(* IEC 61131-3 sources: eCockpitGit/test_project/src/%F%00 Library/%F%Common Functions/%F%Networking/%POU%FB_TCPMultiPlexer, 7 files *)

(* ---- %METH%acceptCycle.st ---- *)
//Called cyclicly to handle incoming connections
// |**Version**|**Author**| **Date** |**Changes**
// | 1         | NSN      | 20-05-22 | Creation
METHOD acceptCycle
VAR
	i			:WORD;
END_VAR
(*%!%__DELIMITER__%!%*)
IF S_nextClosed < S_controllersSize THEN
	//Incoming connection is accepted
	IF S_listenersSize > 0 THEN
		FOR i := 0 TO S_listenersSize - 1 DO
			S_controllers^[S_nextClosed].acceptConnection(listener:=S_listeners^[i]);
		END_FOR
	END_IF
END_IF

(* ---- %METH%closeConnection.st ---- *)
//Called to close and clean up all connections in the multiplexer
// |**Version**|**Author**| **Date** |**Changes**
// | 1         | NSN      | 20-05-22 | Creation
METHOD closeConnection
VAR
	i			:WORD;
END_VAR
(*%!%__DELIMITER__%!%*)
IF S_controllersSize > 0 THEN
	FOR i := 0 TO S_controllersSize - 1 DO
		S_controllers^[i].closeConnection();
	END_FOR
END_IF

(* ---- %METH%initialize.st ---- *)
//Initializes the tcp controller with needed values
// |**Version**|**Author**| **Date** |**Changes**
// | 1         | NSN      | 20-05-22 | Creation
METHOD initialize : SLMResult
VAR_INPUT
	controllers			:POINTER TO ARRAY[0..19] OF FB_TCPController;	//List of controllers to handle connections
	controllersSize		:WORD;											//Size of controller list
	listeners			:POINTER TO ARRAY[0..19] OF TCP.Listener;		//List of listeners to check for incoming connections
	listenersSize		:WORD;											//Size of listener list
END_VAR
VAR
	i					:WORD;
END_VAR
(*%!%__DELIMITER__%!%*)
IF controllers = 0 OR controllersSize = 0 OR listeners = 0 OR listenersSize = 0 THEN
	initialize.success					:=		FALSE;
	initialize.code						:=		ERCodes.FB_TCPMultiPlexer_initialize;
	RETURN;
END_IF
S_controllers							:=		controllers;
S_controllersSize						:=		controllersSize;
FOR i := 0 TO controllersSize - 1 DO
	S_controllers^[i].S_management		:=		THIS^;
	S_controllers^[i].S_index			:=		i;
	IF S_messageEvent <> 0 THEN
		S_controllers^[i].S_message		:=		S_messageEvent;
	END_IF
END_FOR

S_listeners								:=		listeners;
S_listenersSize							:=		listenersSize;

(* ---- %METH%messageCycle.st ---- *)
//Called cyclicly to cause messages to be processed via event system
// |**Version**|**Author**| **Date** |**Changes**
// | 1         | NSN      | 20-05-22 | Creation
METHOD messageCycle
VAR
	i			:WORD;
END_VAR
(*%!%__DELIMITER__%!%*)
IF S_controllersSize > 0 THEN
	FOR i := 0 TO S_controllersSize - 1 DO
		WHILE S_controllers^[i].readyToRecieve DO ; END_WHILE
	END_FOR
END_IF

(* ---- %METH%onClose.st ---- *)
//Called when controller conection is closed
// |**Version**|**Author**| **Date** |**Changes**
// | 1         | NSN      | 20-05-22 | Creation
METHOD onClose
VAR_INPUT
	index			:WORD;				//Index set to controller
END_VAR
VAR_IN_OUT
	controller		:FB_TCPController;	//Controller which is closed
END_VAR
(*%!%__DELIMITER__%!%*)
IF S_nextClosed >= S_controllersSize THEN
	//Next free client is found for next incoming connection
	FOR S_nextClosed := 0 TO S_controllersSize DO
		IF NOT(S_controllers^[S_nextClosed].S_open) THEN
			EXIT;
		END_IF
	END_FOR
END_IF
IF S_management <> 0 THEN
	S_management.onClose(index:=index,controller:=controller);
END_IF
S_amountConnected		:=		S_amountConnected - 1;

(* ---- %METH%onOpen.st ---- *)
//Called when controller conection is opened
// |**Version**|**Author**| **Date** |**Changes**
// | 1         | NSN      | 20-05-22 | Creation
METHOD onOpen: BOOL
VAR_INPUT
	index			:WORD;				//Index set to controller
END_VAR
VAR_IN_OUT
	controller		:FB_TCPController;	//Controller which is closed
END_VAR
(*%!%__DELIMITER__%!%*)
//Next free client is found for next incoming connection
FOR S_nextClosed := 0 TO S_controllersSize DO
	IF NOT(S_controllers^[S_nextClosed].S_open) THEN
		EXIT;
	END_IF
END_FOR
IF S_management <> 0 THEN
	S_management.onOpen(index:=index,controller:=controller);
END_IF
S_amountConnected		:=		S_amountConnected + 1;

(* ---- %METH%sendCycle.st ---- *)
//Called cyclicly to cause messages to be processed via event system
// |**Version**|**Author**| **Date** |**Changes**
// | 1         | NSN      | 20-05-22 | Creation
METHOD sendCycle
VAR
	i			:WORD;
END_VAR
(*%!%__DELIMITER__%!%*)
IF S_controllersSize > 0 THEN
	FOR i := 0 TO S_controllersSize - 1 DO
		S_controllers^[i].cycle();
	END_FOR
END_IF
